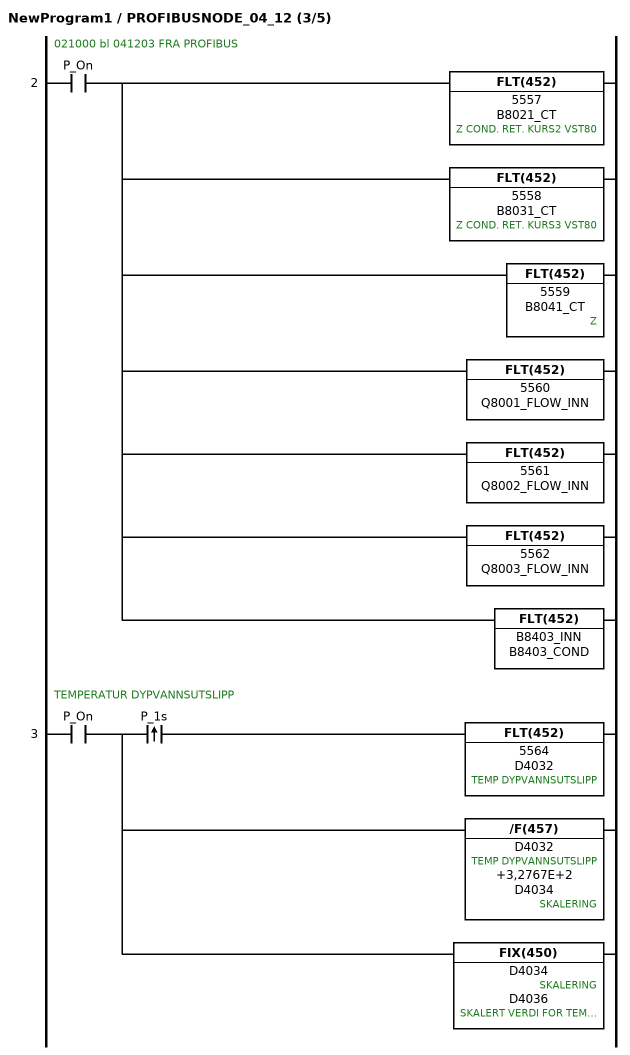
; [picture p1416: NewProgram1 / PROFIBUSNODE_04_12, rungs 2-3]
; rung 2: 021000 bl 041203 FRA PROFIBUS
LD P_On
FLT(452) 5557 B8021_CT  ; Z COND. RET. KURS2 VST80
FLT(452) 5558 B8031_CT  ; Z COND. RET. KURS3 VST80
FLT(452) 5559 B8041_CT  ; Z
FLT(452) 5560 Q8001_FLOW_INN
FLT(452) 5561 Q8002_FLOW_INN
FLT(452) 5562 Q8003_FLOW_INN
FLT(452) B8403_INN B8403_COND
; rung 3: TEMPERATUR DYPVANNSUTSLIPP
LD P_On
OUT TR0
@AND P_1s
FLT(452) 5564 D4032  ; TEMP DYPVANNSUTSLIPP
LD TR0
/F(457) D4032 +3,2767E+2 D4034  ; TEMP DYPVANNSUTSLIPP, SKALERING
FIX(450) D4034 D4036  ; SKALERING, SKALERT VERDI FOR TEMP DYPVANNSUTSLIPP

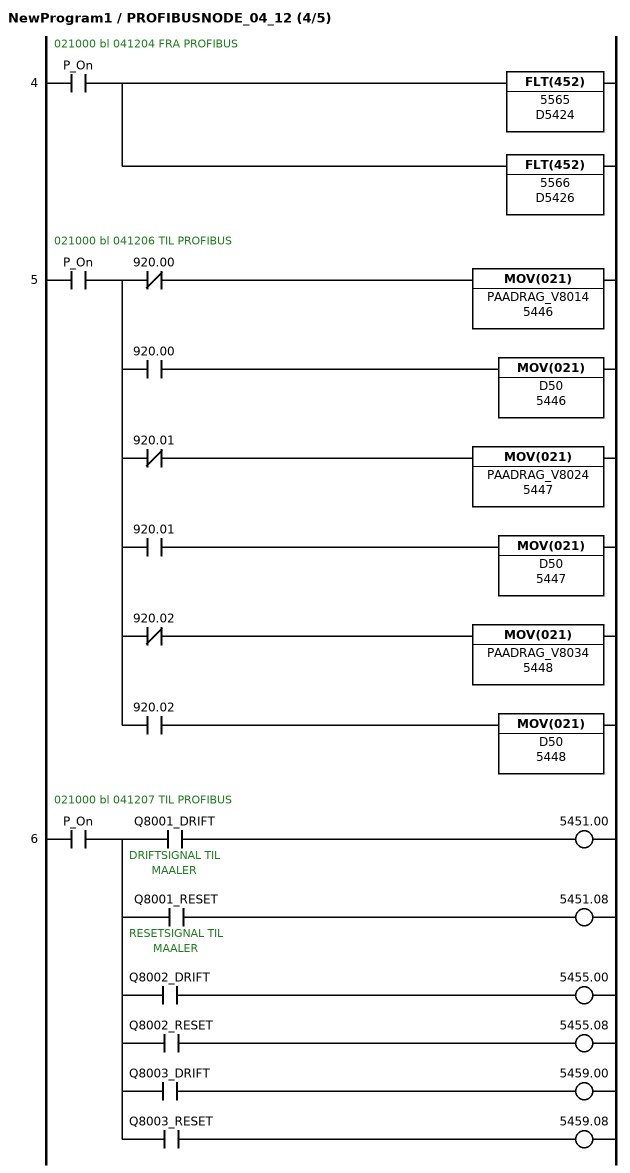
; rung 4: 021000 bl 041204 FRA PROFIBUS
LD P_On
FLT(452) 5565 D5424
FLT(452) 5566 D5426
; rung 5: 021000 bl 041206 TIL PROFIBUS
LD P_On
OUT TR0
ANDNOT 920.00
MOV(021) PAADRAG_V8014 5446
LD TR0
AND 920.00
MOV(021) D50 5446
LD TR0
ANDNOT 920.01
MOV(021) PAADRAG_V8024 5447
LD TR0
AND 920.01
MOV(021) D50 5447
LD TR0
ANDNOT 920.02
MOV(021) PAADRAG_V8034 5448
LD TR0
AND 920.02
MOV(021) D50 5448
; rung 6: 021000 bl 041207 TIL PROFIBUS
LD P_On
OUT TR0
AND Q8001_DRIFT  ; DRIFTSIGNAL TIL MAALER
OUT 5451.00
LD TR0
AND Q8001_RESET  ; RESETSIGNAL TIL MAALER
OUT 5451.08
LD TR0
AND Q8002_DRIFT
OUT 5455.00
LD TR0
AND Q8002_RESET
OUT 5455.08
LD TR0
AND Q8003_DRIFT
OUT 5459.00
LD TR0
AND Q8003_RESET
OUT 5459.08

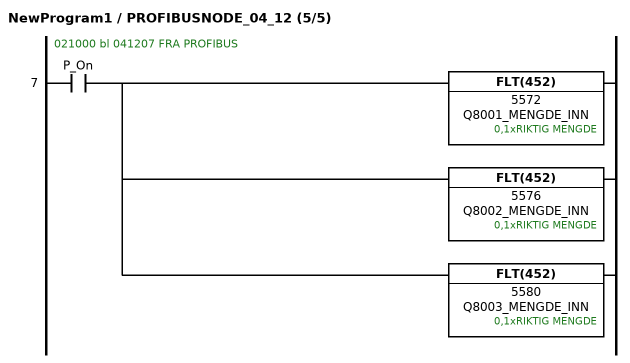
; rung 7: 021000 bl 041207 FRA PROFIBUS
LD P_On
FLT(452) 5572 Q8001_MENGDE_INN  ; 0,1xRIKTIG MENGDE
FLT(452) 5576 Q8002_MENGDE_INN  ; 0,1xRIKTIG MENGDE
FLT(452) 5580 Q8003_MENGDE_INN  ; 0,1xRIKTIG MENGDE
; rung 8: Ingen_kommentar_funnet

### Section PROFIBUSNODE_04_13

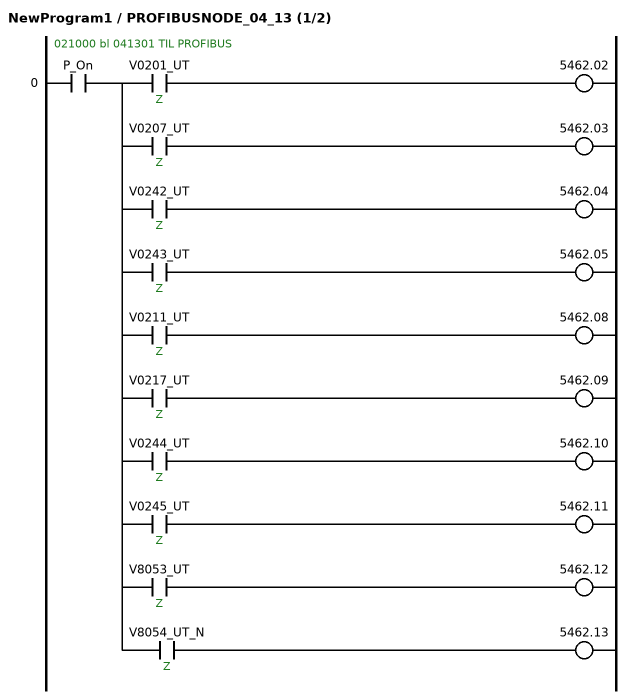
; rung 0: 021000 bl 041301 TIL PROFIBUS
LD P_On
OUT TR0
AND V0201_UT  ; Z
OUT 5462.02
LD TR0
AND V0207_UT  ; Z
OUT 5462.03
LD TR0
AND V0242_UT  ; Z
OUT 5462.04
LD TR0
AND V0243_UT  ; Z
OUT 5462.05
LD TR0
AND V0211_UT  ; Z
OUT 5462.08
LD TR0
AND V0217_UT  ; Z
OUT 5462.09
LD TR0
AND V0244_UT  ; Z
OUT 5462.10
LD TR0
AND V0245_UT  ; Z
OUT 5462.11
LD TR0
AND V8053_UT  ; Z
OUT 5462.12
LD TR0
AND V8054_UT_N  ; Z
OUT 5462.13

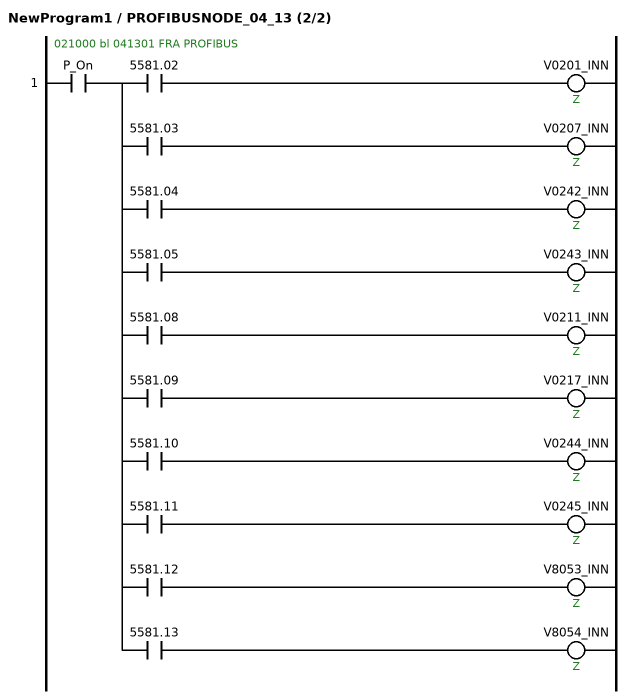
; rung 1: 021000 bl 041301 FRA PROFIBUS
LD P_On
OUT TR0
AND 5581.02
OUT V0201_INN  ; Z
LD TR0
AND 5581.03
OUT V0207_INN  ; Z
LD TR0
AND 5581.04
OUT V0242_INN  ; Z
LD TR0
AND 5581.05
OUT V0243_INN  ; Z
LD TR0
AND 5581.08
OUT V0211_INN  ; Z
LD TR0
AND 5581.09
OUT V0217_INN  ; Z
LD TR0
AND 5581.10
OUT V0244_INN  ; Z
LD TR0
AND 5581.11
OUT V0245_INN  ; Z
LD TR0
AND 5581.12
OUT V8053_INN  ; Z
LD TR0
AND 5581.13
OUT V8054_INN  ; Z
; rung 2: Ingen_kommentar_funnet

### Section PROFIBUSNODE_04_14

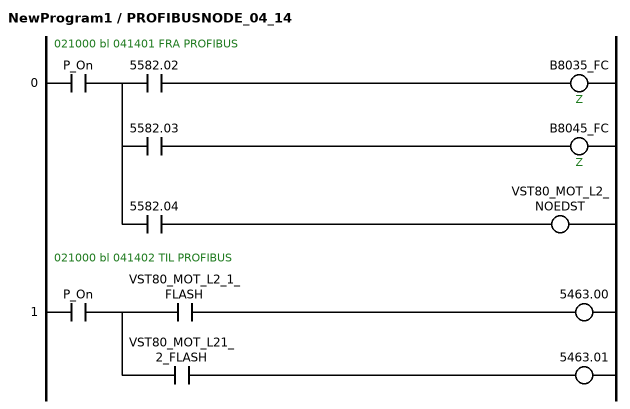
; rung 0: 021000 bl 041401 FRA PROFIBUS
LD P_On
OUT TR0
AND 5582.02
OUT B8035_FC  ; Z
LD TR0
AND 5582.03
OUT B8045_FC  ; Z
LD TR0
AND 5582.04
OUT VST80_MOT_L2_NOEDST
; rung 1: 021000 bl 041402 TIL PROFIBUS
LD P_On
OUT TR0
AND VST80_MOT_L2_1_FLASH
OUT 5463.00
LD TR0
AND VST80_MOT_L21_2_FLASH
OUT 5463.01
; rung 2: Ingen_kommentar_funnet

### Section PROFIBUSNODE_04_15

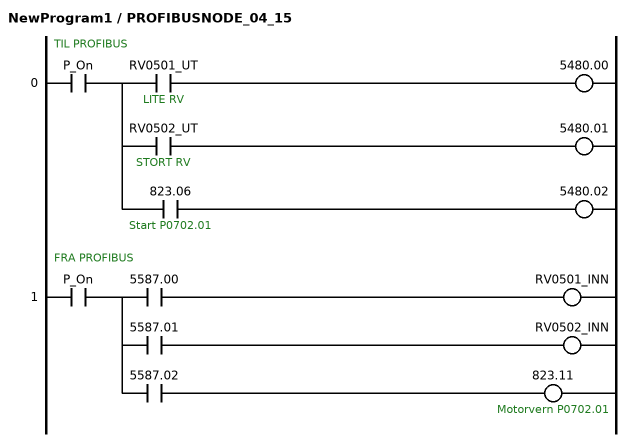
; rung 0: TIL PROFIBUS
LD P_On
OUT TR0
AND RV0501_UT  ; LITE RV
OUT 5480.00
LD TR0
AND RV0502_UT  ; STORT RV
OUT 5480.01
LD TR0
AND 823.06  ; Start P0702.01
OUT 5480.02
; rung 1: FRA PROFIBUS
LD P_On
OUT TR0
AND 5587.00
OUT RV0501_INN
LD TR0
AND 5587.01
OUT RV0502_INN
LD TR0
AND 5587.02
OUT 823.11  ; Motorvern P0702.01
; rung 2: Ingen_kommentar_funnet

### Section PROFIBUSNODE_05_01

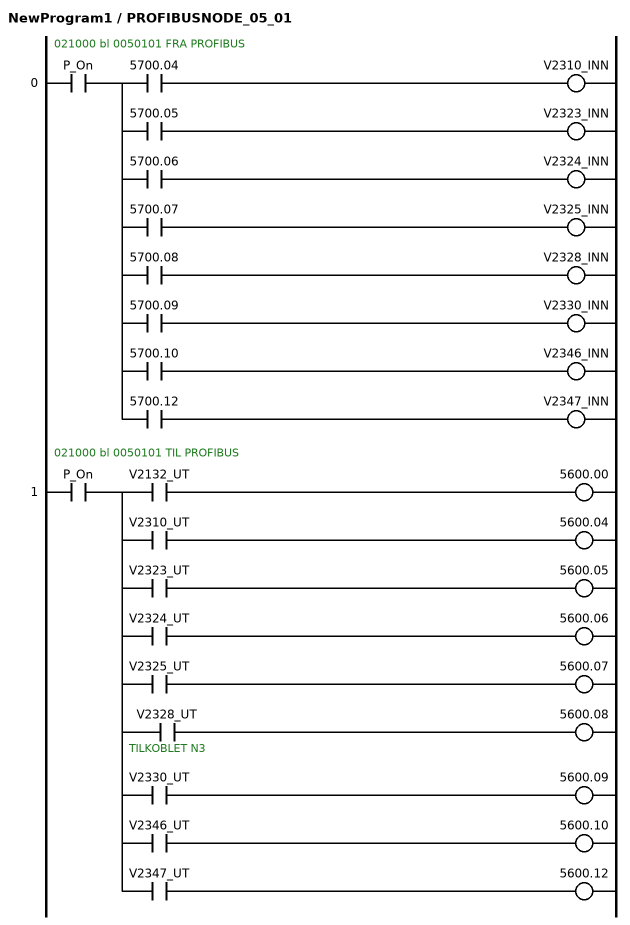
; rung 0: 021000 bl 0050101 FRA PROFIBUS
LD P_On
OUT TR0
AND 5700.04
OUT V2310_INN
LD TR0
AND 5700.05
OUT V2323_INN
LD TR0
AND 5700.06
OUT V2324_INN
LD TR0
AND 5700.07
OUT V2325_INN
LD TR0
AND 5700.08
OUT V2328_INN
LD TR0
AND 5700.09
OUT V2330_INN
LD TR0
AND 5700.10
OUT V2346_INN
LD TR0
AND 5700.12
OUT V2347_INN
; rung 1: 021000 bl 0050101 TIL PROFIBUS
LD P_On
OUT TR0
AND V2132_UT
OUT 5600.00
LD TR0
AND V2310_UT
OUT 5600.04
LD TR0
AND V2323_UT
OUT 5600.05
LD TR0
AND V2324_UT
OUT 5600.06
LD TR0
AND V2325_UT
OUT 5600.07
LD TR0
AND V2328_UT  ; TILKOBLET N3
OUT 5600.08
LD TR0
AND V2330_UT
OUT 5600.09
LD TR0
AND V2346_UT
OUT 5600.10
LD TR0
AND V2347_UT
OUT 5600.12
; rung 2: Ingen_kommentar_funnet

### Section PROFIBUSNODE_05_02

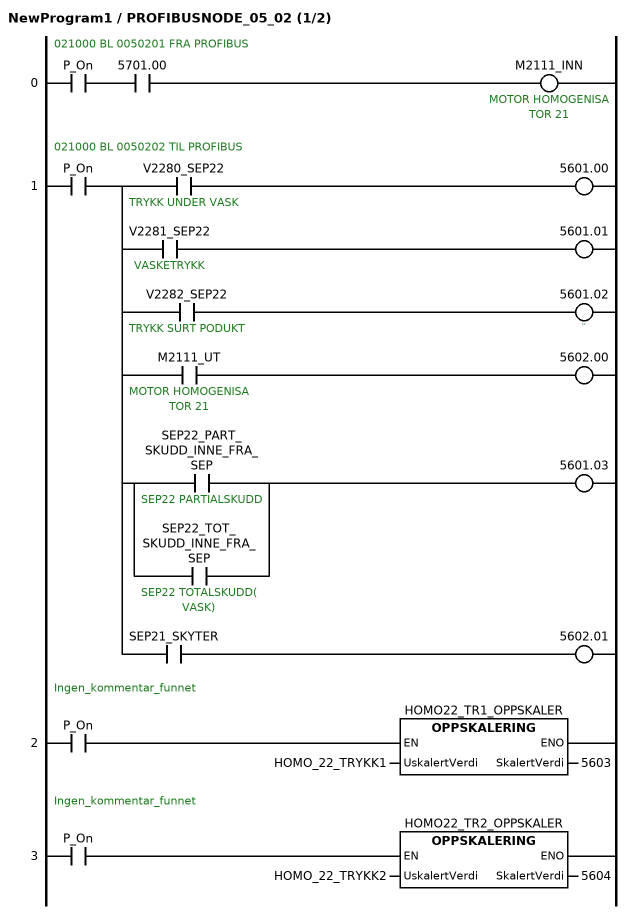
; rung 0: 021000 BL 0050201 FRA PROFIBUS
LD P_On
AND 5701.00
OUT M2111_INN  ; MOTOR HOMOGENISATOR 21
; rung 1: 021000 BL 0050202 TIL PROFIBUS
LD P_On
OUT TR0
AND V2280_SEP22  ; TRYKK UNDER VASK
OUT 5601.00
LD TR0
AND V2281_SEP22  ; VASKETRYKK
OUT 5601.01
LD TR0
AND V2282_SEP22  ; TRYKK SURT PODUKT
OUT 5601.02  ; ¨
LD TR0
AND M2111_UT  ; MOTOR HOMOGENISATOR 21
OUT 5602.00
LD TR0
LD SEP22_PART_SKUDD_INNE_FRA_SEP  ; SEP22 PARTIALSKUDD
OR SEP22_TOT_SKUDD_INNE_FRA_SEP  ; SEP22 TOTALSKUDD(VASK)
ANDLD
OUT 5601.03
LD TR0
AND SEP21_SKYTER
OUT 5602.01
; rung 2: Ingen_kommentar_funnet
LD P_On
CALL HOMO22_TR1_OPPSKALER : OPPSKALERING (UskalertVerdi := HOMO_22_TRYKK1, SkalertVerdi => 5603)
; rung 3: Ingen_kommentar_funnet
LD P_On
CALL HOMO22_TR2_OPPSKALER : OPPSKALERING (UskalertVerdi := HOMO_22_TRYKK2, SkalertVerdi => 5604)

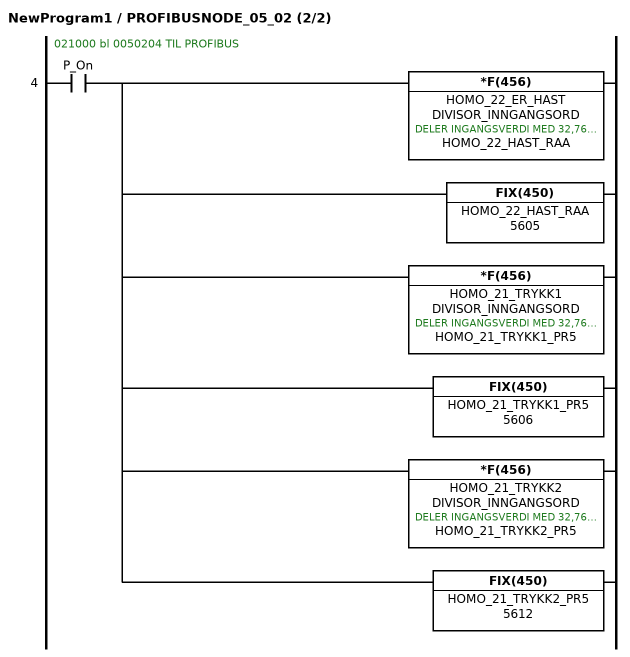
; rung 4: 021000 bl 0050204 TIL PROFIBUS
LD P_On
*F(456) HOMO_22_ER_HAST DIVISOR_INNGANGSORD HOMO_22_HAST_RAA  ; DELER INGANGSVERDI MED 32,760 FOR OMREGNING TIL 0-1000
FIX(450) HOMO_22_HAST_RAA 5605
*F(456) HOMO_21_TRYKK1 DIVISOR_INNGANGSORD HOMO_21_TRYKK1_PR5  ; DELER INGANGSVERDI MED 32,760 FOR OMREGNING TIL 0-1000
FIX(450) HOMO_21_TRYKK1_PR5 5606
*F(456) HOMO_21_TRYKK2 DIVISOR_INNGANGSORD HOMO_21_TRYKK2_PR5  ; DELER INGANGSVERDI MED 32,760 FOR OMREGNING TIL 0-1000
FIX(450) HOMO_21_TRYKK2_PR5 5612
; rung 5: Ingen_kommentar_funnet

### Section PROFIBUSNODE_05_03

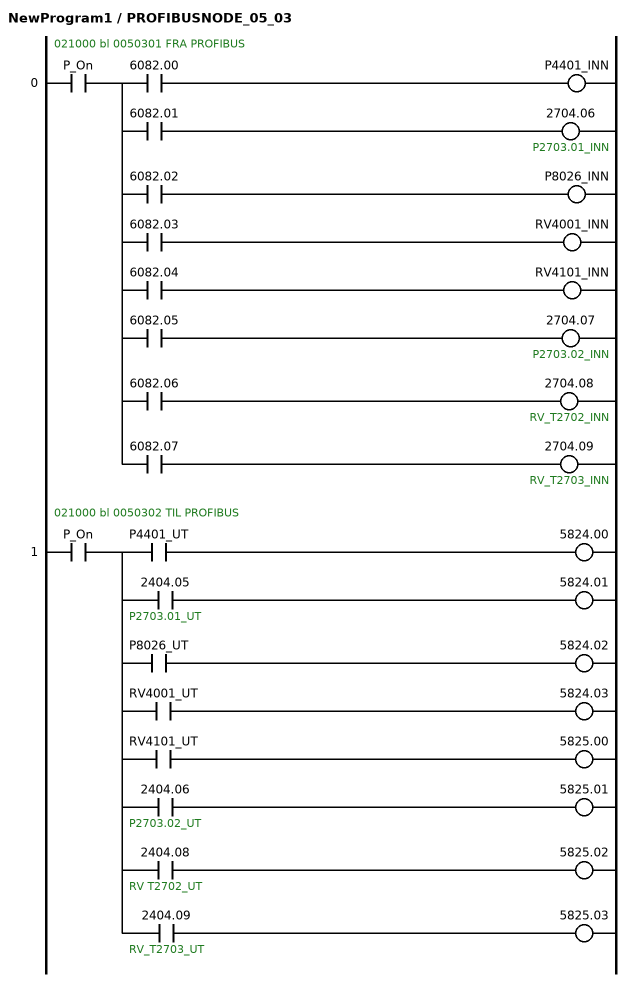
; rung 0: 021000 bl 0050301 FRA PROFIBUS
LD P_On
OUT TR0
AND 6082.00
OUT P4401_INN
LD TR0
AND 6082.01
OUT 2704.06  ; P2703.01_INN
LD TR0
AND 6082.02
OUT P8026_INN
LD TR0
AND 6082.03
OUT RV4001_INN
LD TR0
AND 6082.04
OUT RV4101_INN
LD TR0
AND 6082.05
OUT 2704.07  ; P2703.02_INN
LD TR0
AND 6082.06
OUT 2704.08  ; RV_T2702_INN
LD TR0
AND 6082.07
OUT 2704.09  ; RV_T2703_INN
; rung 1: 021000 bl 0050302 TIL PROFIBUS
LD P_On
OUT TR0
AND P4401_UT
OUT 5824.00
LD TR0
AND 2404.05  ; P2703.01_UT
OUT 5824.01
LD TR0
AND P8026_UT
OUT 5824.02
LD TR0
AND RV4001_UT
OUT 5824.03
LD TR0
AND RV4101_UT
OUT 5825.00
LD TR0
AND 2404.06  ; P2703.02_UT
OUT 5825.01
LD TR0
AND 2404.08  ; RV T2702_UT
OUT 5825.02
LD TR0
AND 2404.09  ; RV_T2703_UT
OUT 5825.03
; rung 2: Ingen_kommentar_funnet

### Section PROFIBUSNODE_05_05

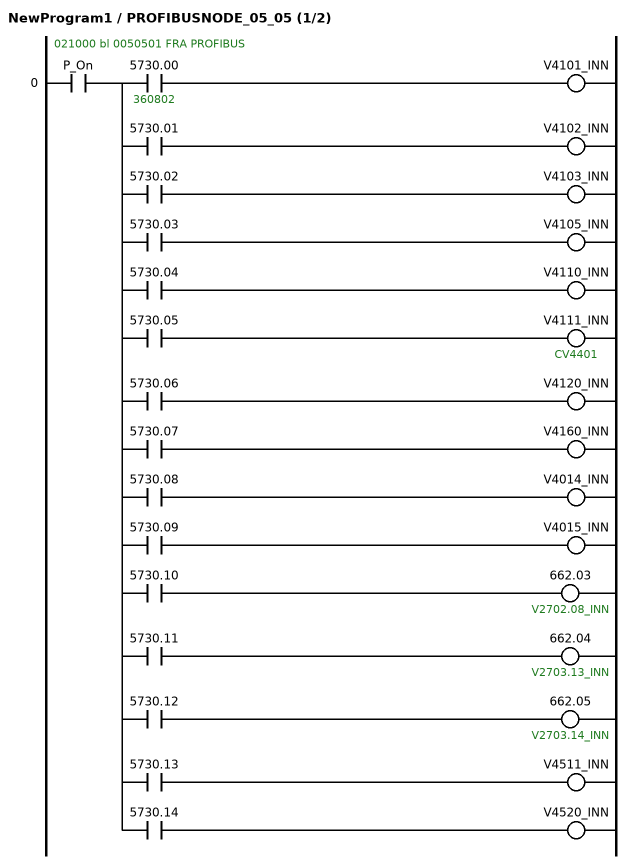
; rung 0: 021000 bl 0050501 FRA PROFIBUS
LD P_On
OUT TR0
AND 5730.00  ; 360802
OUT V4101_INN
LD TR0
AND 5730.01
OUT V4102_INN
LD TR0
AND 5730.02
OUT V4103_INN
LD TR0
AND 5730.03
OUT V4105_INN
LD TR0
AND 5730.04
OUT V4110_INN
LD TR0
AND 5730.05
OUT V4111_INN  ; CV4401
LD TR0
AND 5730.06
OUT V4120_INN
LD TR0
AND 5730.07
OUT V4160_INN
LD TR0
AND 5730.08
OUT V4014_INN
LD TR0
AND 5730.09
OUT V4015_INN
LD TR0
AND 5730.10
OUT 662.03  ; V2702.08_INN
LD TR0
AND 5730.11
OUT 662.04  ; V2703.13_INN
LD TR0
AND 5730.12
OUT 662.05  ; V2703.14_INN
LD TR0
AND 5730.13
OUT V4511_INN
LD TR0
AND 5730.14
OUT V4520_INN

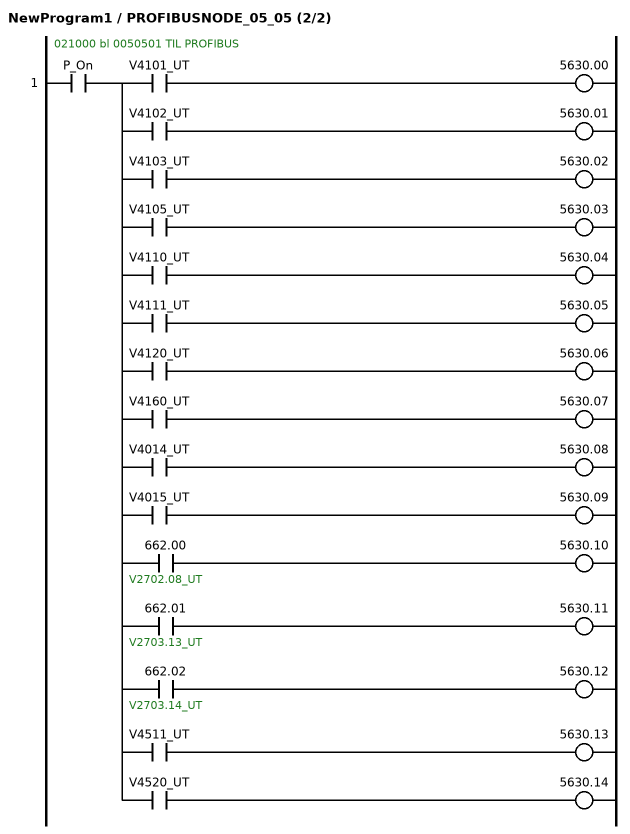
; rung 1: 021000 bl 0050501 TIL PROFIBUS
LD P_On
OUT TR0
AND V4101_UT
OUT 5630.00
LD TR0
AND V4102_UT
OUT 5630.01
LD TR0
AND V4103_UT
OUT 5630.02
LD TR0
AND V4105_UT
OUT 5630.03
LD TR0
AND V4110_UT
OUT 5630.04
LD TR0
AND V4111_UT
OUT 5630.05
LD TR0
AND V4120_UT
OUT 5630.06
LD TR0
AND V4160_UT
OUT 5630.07
LD TR0
AND V4014_UT
OUT 5630.08
LD TR0
AND V4015_UT
OUT 5630.09
LD TR0
AND 662.00  ; V2702.08_UT
OUT 5630.10
LD TR0
AND 662.01  ; V2703.13_UT
OUT 5630.11
LD TR0
AND 662.02  ; V2703.14_UT
OUT 5630.12
LD TR0
AND V4511_UT
OUT 5630.13
LD TR0
AND V4520_UT
OUT 5630.14
; rung 2: Ingen_kommentar_funnet

### Section PROFIBUSNODE_05_04

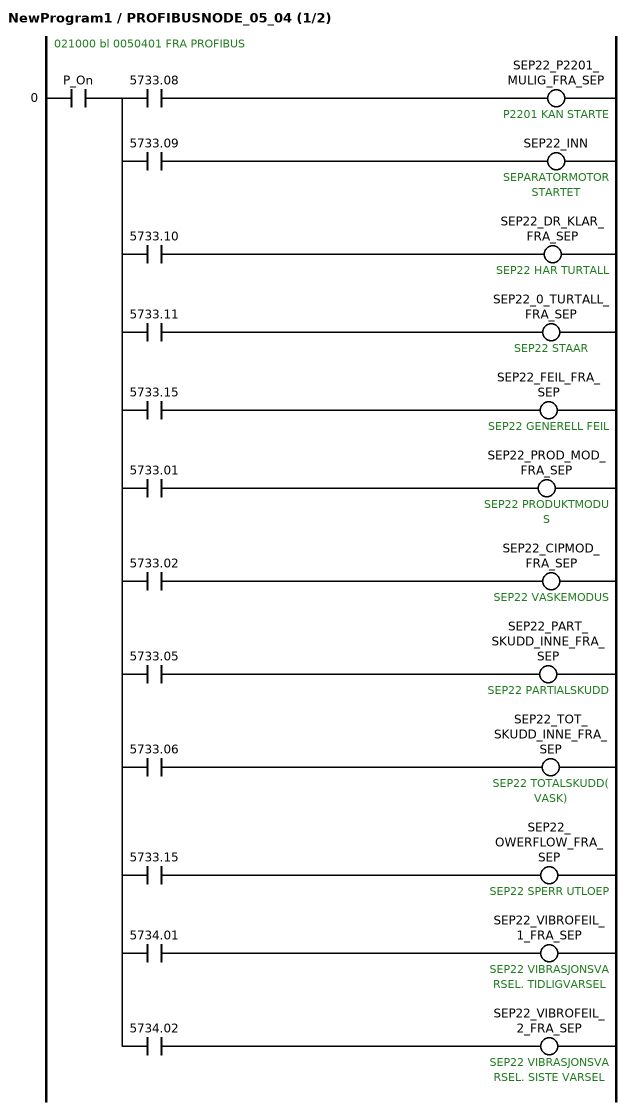
; rung 0: 021000 bl 0050401 FRA PROFIBUS
LD P_On
OUT TR0
AND 5733.08
OUT SEP22_P2201_MULIG_FRA_SEP  ; P2201 KAN STARTE
LD TR0
AND 5733.09
OUT SEP22_INN  ; SEPARATORMOTOR STARTET
LD TR0
AND 5733.10
OUT SEP22_DR_KLAR_FRA_SEP  ; SEP22 HAR TURTALL
LD TR0
AND 5733.11
OUT SEP22_0_TURTALL_FRA_SEP  ; SEP22 STAAR
LD TR0
AND 5733.15
OUT SEP22_FEIL_FRA_SEP  ; SEP22 GENERELL FEIL
LD TR0
AND 5733.01
OUT SEP22_PROD_MOD_FRA_SEP  ; SEP22 PRODUKTMODUS
LD TR0
AND 5733.02
OUT SEP22_CIPMOD_FRA_SEP  ; SEP22 VASKEMODUS
LD TR0
AND 5733.05
OUT SEP22_PART_SKUDD_INNE_FRA_SEP  ; SEP22 PARTIALSKUDD
LD TR0
AND 5733.06
OUT SEP22_TOT_SKUDD_INNE_FRA_SEP  ; SEP22 TOTALSKUDD(VASK)
LD TR0
AND 5733.15
OUT SEP22_OWERFLOW_FRA_SEP  ; SEP22 SPERR UTLOEP
LD TR0
AND 5734.01
OUT SEP22_VIBROFEIL_1_FRA_SEP  ; SEP22 VIBRASJONSVARSEL. TIDLIGVARSEL
LD TR0
AND 5734.02
OUT SEP22_VIBROFEIL_2_FRA_SEP  ; SEP22 VIBRASJONSVARSEL. SISTE VARSEL

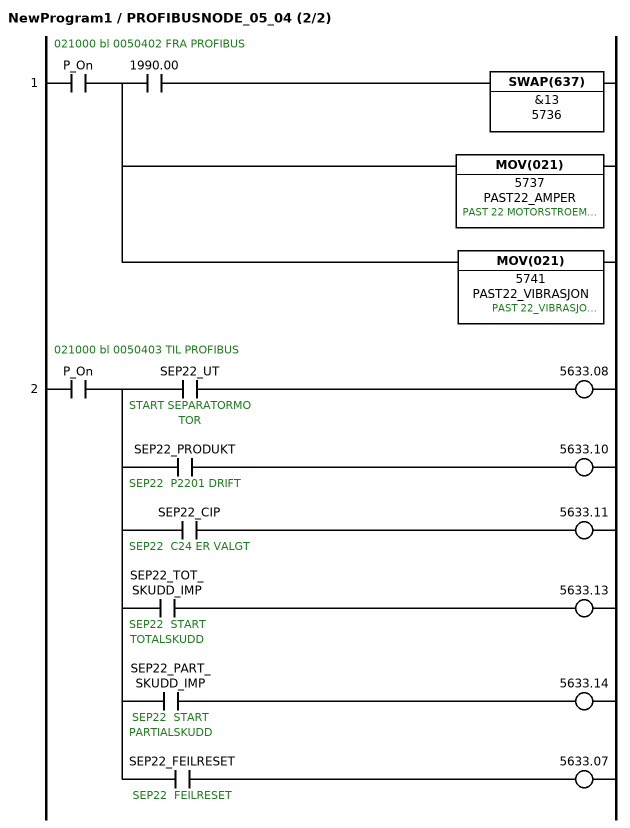
; rung 1: 021000 bl 0050402 FRA PROFIBUS
LD P_On
OUT TR0
AND 1990.00
SWAP(637) &13 5736
LD TR0
MOV(021) 5737 PAST22_AMPER  ; PAST 22 MOTORSTROEM. 1000=100,0 AMP
MOV(021) 5741 PAST22_VIBRASJON  ; PAST 22_VIBRASJON 2000=20,00mm/S
; rung 2: 021000 bl 0050403 TIL PROFIBUS
LD P_On
OUT TR0
AND SEP22_UT  ; START SEPARATORMOTOR
OUT 5633.08
LD TR0
AND SEP22_PRODUKT  ; SEP22  P2201 DRIFT
OUT 5633.10
LD TR0
AND SEP22_CIP  ; SEP22  C24 ER VALGT
OUT 5633.11
LD TR0
AND SEP22_TOT_SKUDD_IMP  ; SEP22  START TOTALSKUDD
OUT 5633.13
LD TR0
AND SEP22_PART_SKUDD_IMP  ; SEP22  START PARTIALSKUDD
OUT 5633.14
LD TR0
AND SEP22_FEILRESET  ; SEP22  FEILRESET
OUT 5633.07
; rung 3: Ingen_kommentar_funnet

### Section PROFIBUSNODE_05_06

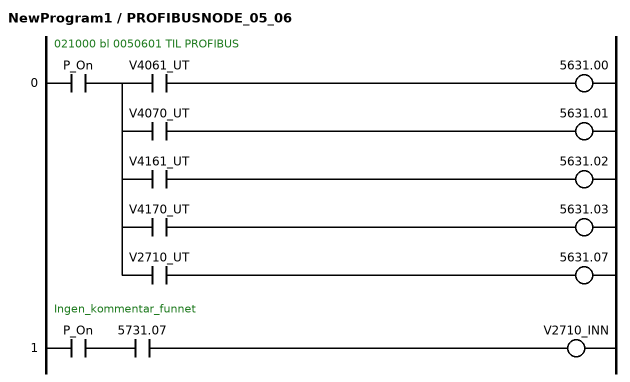
; rung 0: 021000 bl 0050601 TIL PROFIBUS
LD P_On
OUT TR0
AND V4061_UT
OUT 5631.00
LD TR0
AND V4070_UT
OUT 5631.01
LD TR0
AND V4161_UT
OUT 5631.02
LD TR0
AND V4170_UT
OUT 5631.03
LD TR0
AND V2710_UT
OUT 5631.07
; rung 1: Ingen_kommentar_funnet
LD P_On
AND 5731.07
OUT V2710_INN
; rung 2: Ingen_kommentar_funnet

### Section PROFIBUSNODE_05_07

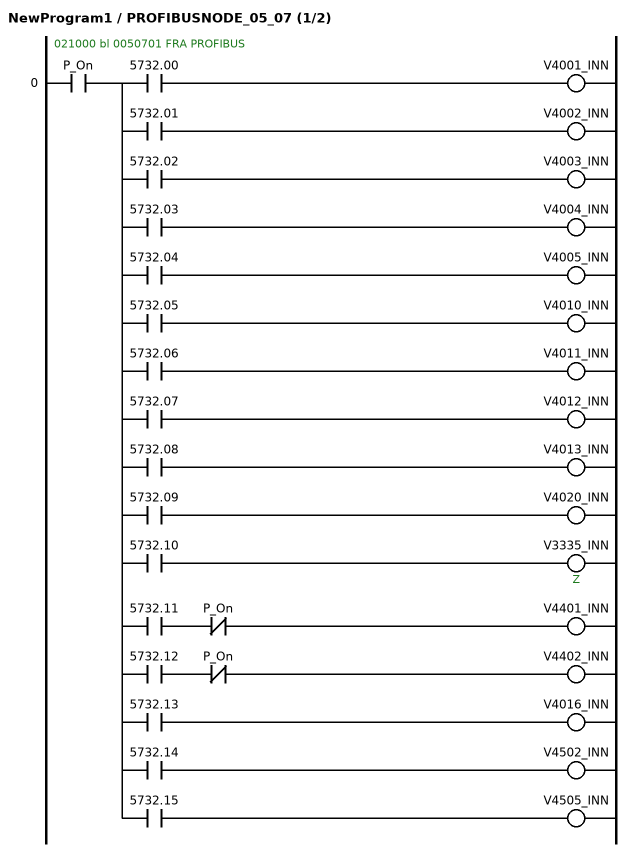
; rung 0: 021000 bl 0050701 FRA PROFIBUS
LD P_On
OUT TR0
AND 5732.00
OUT V4001_INN
LD TR0
AND 5732.01
OUT V4002_INN
LD TR0
AND 5732.02
OUT V4003_INN
LD TR0
AND 5732.03
OUT V4004_INN
LD TR0
AND 5732.04
OUT V4005_INN
LD TR0
AND 5732.05
OUT V4010_INN
LD TR0
AND 5732.06
OUT V4011_INN
LD TR0
AND 5732.07
OUT V4012_INN
LD TR0
AND 5732.08
OUT V4013_INN
LD TR0
AND 5732.09
OUT V4020_INN
LD TR0
AND 5732.10
OUT V3335_INN  ; Z
LD TR0
AND 5732.11
ANDNOT P_On
OUT V4401_INN
LD TR0
AND 5732.12
ANDNOT P_On
OUT V4402_INN
LD TR0
AND 5732.13
OUT V4016_INN
LD TR0
AND 5732.14
OUT V4502_INN
LD TR0
AND 5732.15
OUT V4505_INN

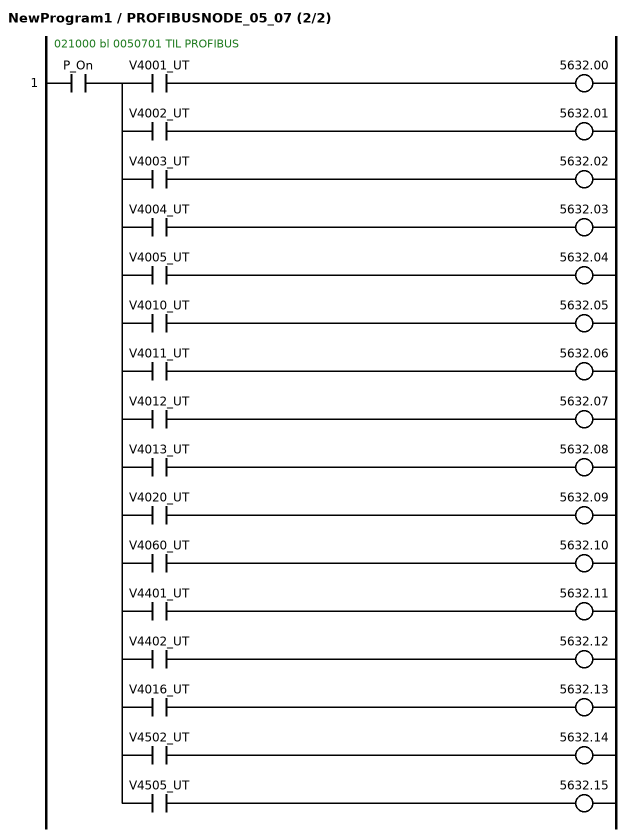
; rung 1: 021000 bl 0050701 TIL PROFIBUS
LD P_On
OUT TR0
AND V4001_UT
OUT 5632.00
LD TR0
AND V4002_UT
OUT 5632.01
LD TR0
AND V4003_UT
OUT 5632.02
LD TR0
AND V4004_UT
OUT 5632.03
LD TR0
AND V4005_UT
OUT 5632.04
LD TR0
AND V4010_UT
OUT 5632.05
LD TR0
AND V4011_UT
OUT 5632.06
LD TR0
AND V4012_UT
OUT 5632.07
LD TR0
AND V4013_UT
OUT 5632.08
LD TR0
AND V4020_UT
OUT 5632.09
LD TR0
AND V4060_UT
OUT 5632.10
LD TR0
AND V4401_UT
OUT 5632.11
LD TR0
AND V4402_UT
OUT 5632.12
LD TR0
AND V4016_UT
OUT 5632.13
LD TR0
AND V4502_UT
OUT 5632.14
LD TR0
AND V4505_UT
OUT 5632.15
; rung 2: Ingen_kommentar_funnet

### Section PROFIBUSNODE_05_08

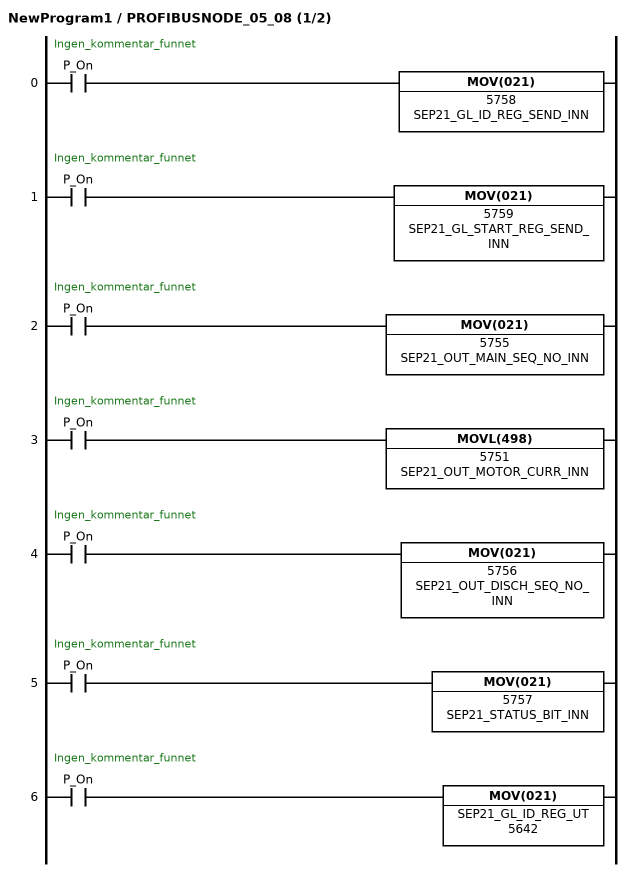
; rung 0: Ingen_kommentar_funnet
LD P_On
MOV(021) 5758 SEP21_GL_ID_REG_SEND_INN
; rung 1: Ingen_kommentar_funnet
LD P_On
MOV(021) 5759 SEP21_GL_START_REG_SEND_INN
; rung 2: Ingen_kommentar_funnet
LD P_On
MOV(021) 5755 SEP21_OUT_MAIN_SEQ_NO_INN
; rung 3: Ingen_kommentar_funnet
LD P_On
MOVL(498) 5751 SEP21_OUT_MOTOR_CURR_INN
; rung 4: Ingen_kommentar_funnet
LD P_On
MOV(021) 5756 SEP21_OUT_DISCH_SEQ_NO_INN
; rung 5: Ingen_kommentar_funnet
LD P_On
MOV(021) 5757 SEP21_STATUS_BIT_INN
; rung 6: Ingen_kommentar_funnet
LD P_On
MOV(021) SEP21_GL_ID_REG_UT 5642

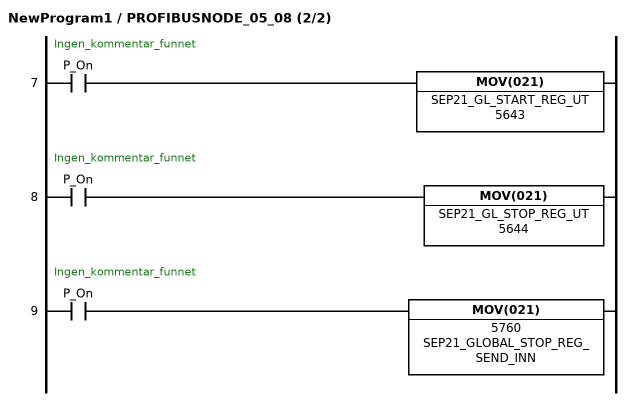
; rung 7: Ingen_kommentar_funnet
LD P_On
MOV(021) SEP21_GL_START_REG_UT 5643
; rung 8: Ingen_kommentar_funnet
LD P_On
MOV(021) SEP21_GL_STOP_REG_UT 5644
; rung 9: Ingen_kommentar_funnet
LD P_On
MOV(021) 5760 SEP21_GLOBAL_STOP_REG_SEND_INN
; rung 10: Ingen_kommentar_funnet

### Section PROFIBUSNODE_05_09

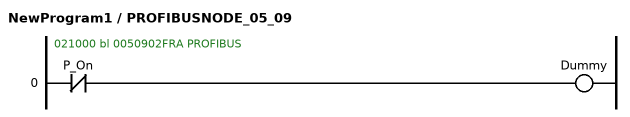
; rung 0: 021000 bl 0050902FRA PROFIBUS
LDNOT P_On
OUT Dummy
; rung 1: Ingen_kommentar_funnet

### Section PROFIBUSNODE_05_10

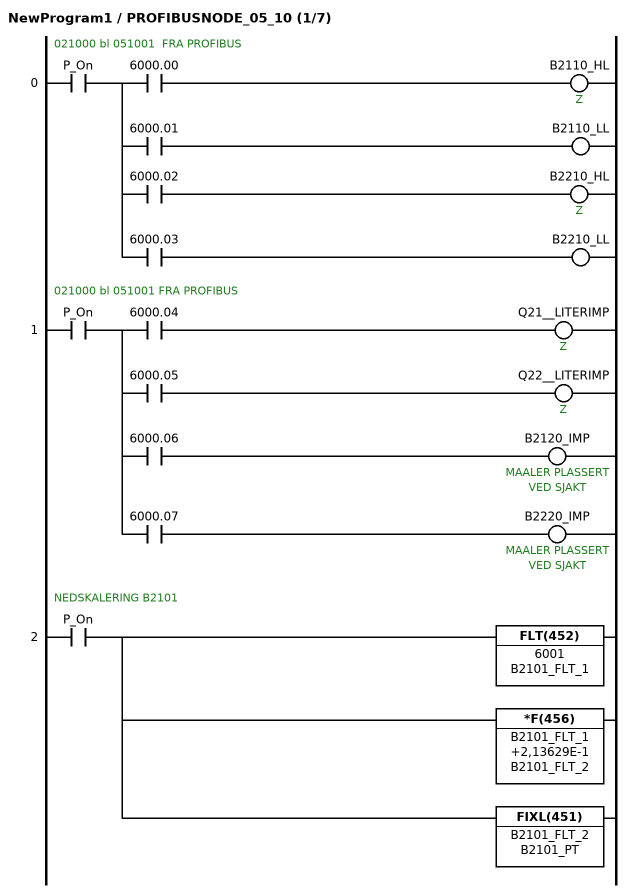
; rung 0: 021000 bl 051001  FRA PROFIBUS
LD P_On
OUT TR0
AND 6000.00
OUT B2110_HL  ; Z
LD TR0
AND 6000.01
OUT B2110_LL
LD TR0
AND 6000.02
OUT B2210_HL  ; Z
LD TR0
AND 6000.03
OUT B2210_LL
; rung 1: 021000 bl 051001 FRA PROFIBUS
LD P_On
OUT TR0
AND 6000.04
OUT Q21__LITERIMP  ; Z
LD TR0
AND 6000.05
OUT Q22__LITERIMP  ; Z
LD TR0
AND 6000.06
OUT B2120_IMP  ; MAALER PLASSERT VED SJAKT
LD TR0
AND 6000.07
OUT B2220_IMP  ; MAALER PLASSERT VED SJAKT
; rung 2: NEDSKALERING B2101
LD P_On
FLT(452) 6001 B2101_FLT_1
*F(456) B2101_FLT_1 +2,13629E-1 B2101_FLT_2
FIXL(451) B2101_FLT_2 B2101_PT

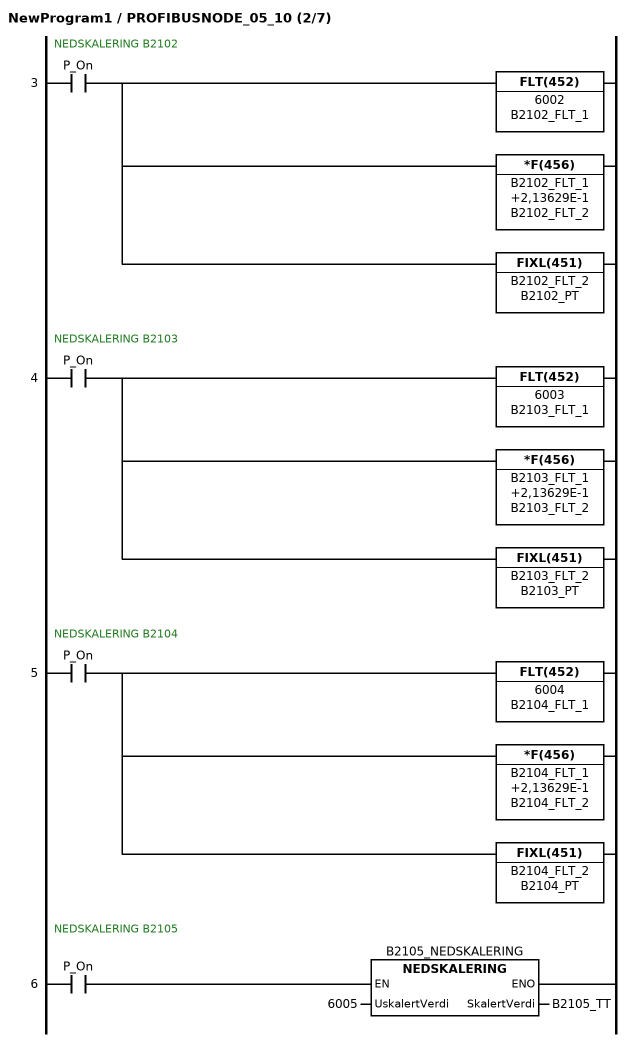
; rung 3: NEDSKALERING B2102
LD P_On
FLT(452) 6002 B2102_FLT_1
*F(456) B2102_FLT_1 +2,13629E-1 B2102_FLT_2
FIXL(451) B2102_FLT_2 B2102_PT
; rung 4: NEDSKALERING B2103
LD P_On
FLT(452) 6003 B2103_FLT_1
*F(456) B2103_FLT_1 +2,13629E-1 B2103_FLT_2
FIXL(451) B2103_FLT_2 B2103_PT
; rung 5: NEDSKALERING B2104
LD P_On
FLT(452) 6004 B2104_FLT_1
*F(456) B2104_FLT_1 +2,13629E-1 B2104_FLT_2
FIXL(451) B2104_FLT_2 B2104_PT
; rung 6: NEDSKALERING B2105
LD P_On
CALL B2105_NEDSKALERING : NEDSKALERING (UskalertVerdi := 6005, SkalertVerdi => B2105_TT)

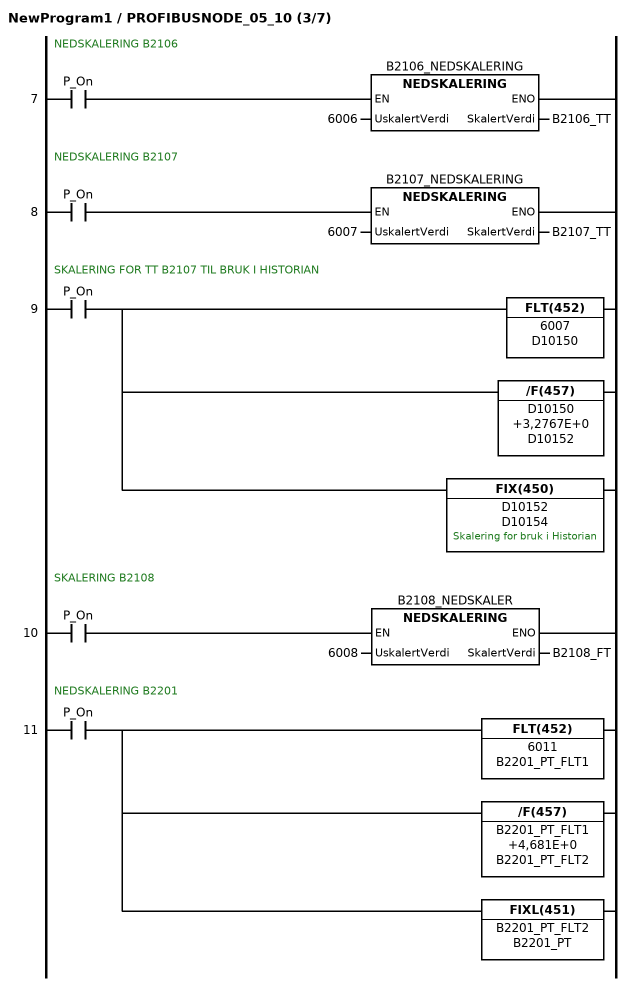
; rung 7: NEDSKALERING B2106
LD P_On
CALL B2106_NEDSKALERING : NEDSKALERING (UskalertVerdi := 6006, SkalertVerdi => B2106_TT)
; rung 8: NEDSKALERING B2107
LD P_On
CALL B2107_NEDSKALERING : NEDSKALERING (UskalertVerdi := 6007, SkalertVerdi => B2107_TT)
; rung 9: SKALERING FOR TT B2107 TIL BRUK I HISTORIAN
LD P_On
FLT(452) 6007 D10150
/F(457) D10150 +3,2767E+0 D10152
FIX(450) D10152 D10154  ; Skalering for bruk i Historian
; rung 10: SKALERING B2108
LD P_On
CALL B2108_NEDSKALER : NEDSKALERING (UskalertVerdi := 6008, SkalertVerdi => B2108_FT)
; rung 11: NEDSKALERING B2201
LD P_On
FLT(452) 6011 B2201_PT_FLT1
/F(457) B2201_PT_FLT1 +4,681E+0 B2201_PT_FLT2
FIXL(451) B2201_PT_FLT2 B2201_PT

